// TIA Portal V19 export
FUNCTION "FC70_Counter" : Void   // FC2, LAD
{ S7_Optimized_Access := 'TRUE' }
// stored: IsIECCheckEnabled true, SetENOAutomatically false
BEGIN

REGION Network 1: Running time counter
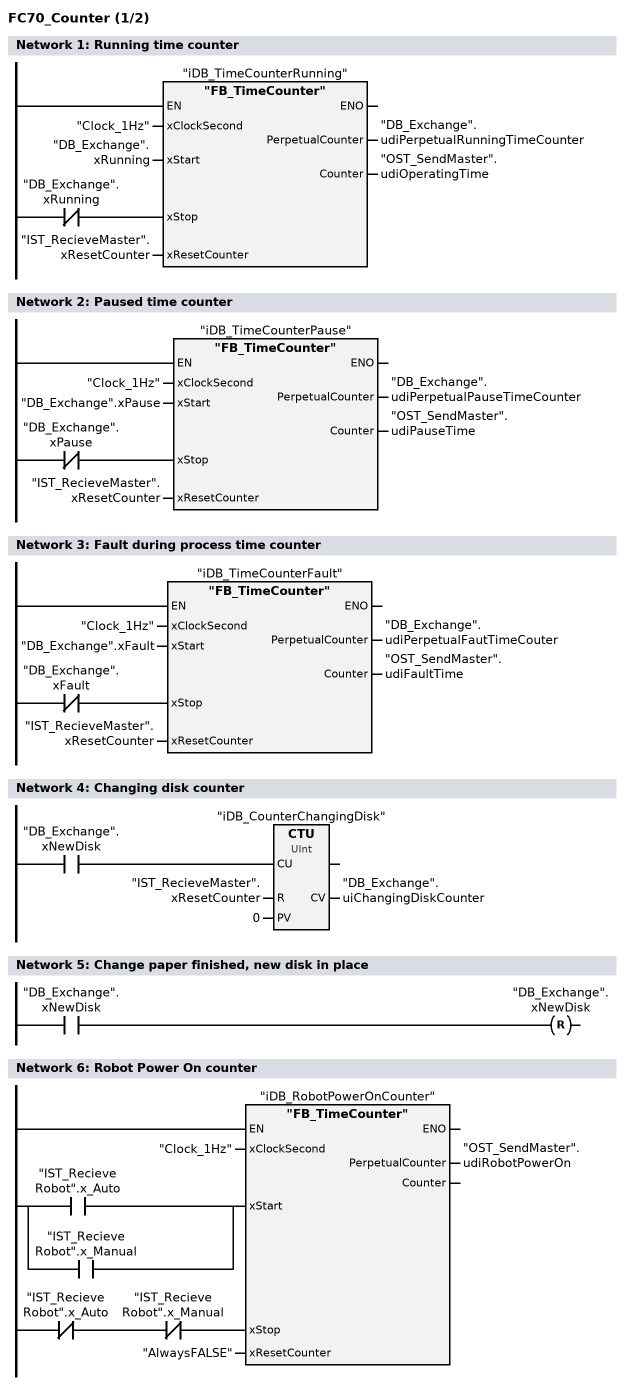
   RUNG wire#powerrail
      "iDB_TimeCounterRunning"(xStop := wire#w1, xClockSecond := "Clock_1Hz", xStart := "DB_Exchange".xRunning, xResetCounter := "IST_RecieveMaster".xResetCounter, PerpetualCounter => "DB_Exchange".udiPerpetualRunningTimeCounter, "Counter" => "OST_SendMaster".udiOperatingTime)
   END_RUNG
   RUNG wire#powerrail
      I_Contact( "DB_Exchange".xRunning )
   END_RUNG wire#w1
   // the same network as SCL:
   "iDB_TimeCounterRunning"(xClockSecond := "Clock_1Hz",   // "FB_TimeCounter"
                           xStart := "DB_Exchange".xRunning,
                           xStop := NOT "DB_Exchange".xRunning,
                           xResetCounter := "IST_RecieveMaster".xResetCounter,
                           PerpetualCounter => "DB_Exchange".udiPerpetualRunningTimeCounter,
                           "Counter" => "OST_SendMaster".udiOperatingTime);
END_REGION

REGION Network 2: Paused time counter
   RUNG wire#powerrail
      "iDB_TimeCounterPause"(xStop := wire#w1, xClockSecond := "Clock_1Hz", xStart := "DB_Exchange".xPause, xResetCounter := "IST_RecieveMaster".xResetCounter, PerpetualCounter => "DB_Exchange".udiPerpetualPauseTimeCounter, "Counter" => "OST_SendMaster".udiPauseTime)
   END_RUNG
   RUNG wire#powerrail
      I_Contact( "DB_Exchange".xPause )
   END_RUNG wire#w1
   // the same network as SCL:
   "iDB_TimeCounterPause"(xClockSecond := "Clock_1Hz",   // "FB_TimeCounter"
                          xStart := "DB_Exchange".xPause,
                          xStop := NOT "DB_Exchange".xPause,
                          xResetCounter := "IST_RecieveMaster".xResetCounter,
                          PerpetualCounter => "DB_Exchange".udiPerpetualPauseTimeCounter,
                          "Counter" => "OST_SendMaster".udiPauseTime);
END_REGION

REGION Network 3: Fault during process time counter
   RUNG wire#powerrail
      "iDB_TimeCounterFault"(xStop := wire#w1, xClockSecond := "Clock_1Hz", xStart := "DB_Exchange".xFault, xResetCounter := "IST_RecieveMaster".xResetCounter, PerpetualCounter => "DB_Exchange".udiPerpetualFautTimeCouter, "Counter" => "OST_SendMaster".udiFaultTime)
   END_RUNG
   RUNG wire#powerrail
      I_Contact( "DB_Exchange".xFault )
   END_RUNG wire#w1
   // the same network as SCL:
   "iDB_TimeCounterFault"(xClockSecond := "Clock_1Hz",   // "FB_TimeCounter"
                          xStart := "DB_Exchange".xFault,
                          xStop := NOT "DB_Exchange".xFault,
                          xResetCounter := "IST_RecieveMaster".xResetCounter,
                          PerpetualCounter => "DB_Exchange".udiPerpetualFautTimeCouter,
                          "Counter" => "OST_SendMaster".udiFaultTime);
END_REGION

REGION Network 4: Changing disk counter
   RUNG wire#powerrail
      Contact( "DB_Exchange".xNewDisk )
      { S7_Templates := "value_type := UInt" } "iDB_CounterChangingDisk".CTU(r := "IST_RecieveMaster".xResetCounter, pv := 0, cv => "DB_Exchange".uiChangingDiskCounter)
   END_RUNG
   // the same network as SCL:
   "iDB_CounterChangingDisk".CTU(CU := "DB_Exchange".xNewDisk,
                           R := "IST_RecieveMaster".xResetCounter,
                           PV := 0,
                           CV => "DB_Exchange".uiChangingDiskCounter);
END_REGION

REGION Network 5: Change paper finished, new disk in place
   RUNG wire#powerrail
      Contact( "DB_Exchange".xNewDisk )
      R_Coil( "DB_Exchange".xNewDisk )
   END_RUNG
   // the same network as SCL:
   IF "DB_Exchange".xNewDisk THEN "DB_Exchange".xNewDisk := FALSE; END_IF;
END_REGION

REGION Network 6: Robot Power On counter
   RUNG wire#powerrail
      "iDB_RobotPowerOnCounter"(xStart := wire#w1, xStop := wire#w2, xClockSecond := "Clock_1Hz", xResetCounter := "AlwaysFALSE", PerpetualCounter => "OST_SendMaster".udiRobotPowerOn, "Counter" =>)
   END_RUNG
   RUNG wire#powerrail
      Contact( "IST_RecieveRobot".x_Auto )
   END_RUNG wire#w1
   RUNG wire#powerrail
      Contact( "IST_RecieveRobot".x_Manual )
   END_RUNG wire#w1
   RUNG wire#powerrail
      I_Contact( "IST_RecieveRobot".x_Auto )
      I_Contact( "IST_RecieveRobot".x_Manual )
   END_RUNG wire#w2
   // the same network as SCL:
   "iDB_RobotPowerOnCounter"(xClockSecond := "Clock_1Hz",   // "FB_TimeCounter"
                           xStart := "IST_RecieveRobot".x_Auto OR "IST_RecieveRobot".x_Manual,
                           xStop := NOT "IST_RecieveRobot".x_Auto AND NOT "IST_RecieveRobot".x_Manual,
                           xResetCounter := "AlwaysFALSE",
                           PerpetualCounter => "OST_SendMaster".udiRobotPowerOn);
END_REGION

REGION Network 7: Robot Drive On counter
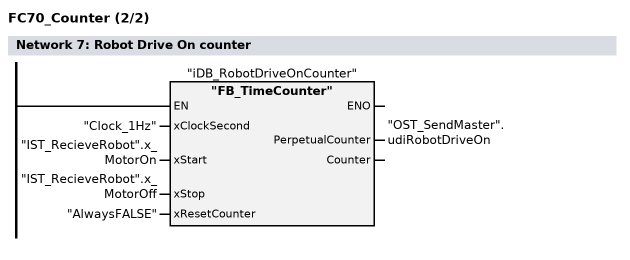
   RUNG wire#powerrail
      "iDB_RobotDriveOnCounter"(xClockSecond := "Clock_1Hz", xStart := "IST_RecieveRobot".x_MotorOn, xStop := "IST_RecieveRobot".x_MotorOff, xResetCounter := "AlwaysFALSE", PerpetualCounter => "OST_SendMaster".udiRobotDriveOn, "Counter" =>)
   END_RUNG
   // the same network as SCL:
   "iDB_RobotDriveOnCounter"(xClockSecond := "Clock_1Hz",   // "FB_TimeCounter"
                           xStart := "IST_RecieveRobot".x_MotorOn,
                           xStop := "IST_RecieveRobot".x_MotorOff,
                           xResetCounter := "AlwaysFALSE",
                           PerpetualCounter => "OST_SendMaster".udiRobotDriveOn);
END_REGION
END_FUNCTION
